TYPE ST_MACHINE :
STRUCT
	
	sName						: STRING;
	
	bMachine					: ARRAY [1..3] OF BOOL;
		
	bHeightTest 				: BOOL;
	bVisionTest					: BOOL;
	bLeakTest					: BOOL;
	bPuckLocker				: BOOL; //Renan Added 10Jul26 - Puck Locker

END_STRUCT
END_TYPE

(* stored: Version 1.1.0.1, ProductVersion 3.1.4026.17
   DUT ST_MACHINE: Id {07cde51d-2827-4fa0-b86f-854c260785fb} *)
